FUNCTION_BLOCK MultiIOthersVlvStatus (* Composite Function Block Type *)
  (* Standard: 61499-2 *)
  (* Version 0.0, 8/28/2026, Schneider Electric, template *)
  PACKAGE SE.Nereda;
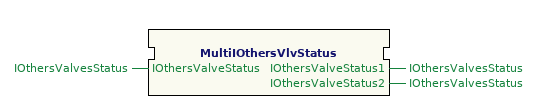
  SOCKETS
    IOthersValveStatus : IOthersValvesStatus;
  END_SOCKETS
  PLUGS
    IOthersValveStatus1 : IOthersValvesStatus;
    IOthersValveStatus2 : IOthersValvesStatus;
  END_PLUGS
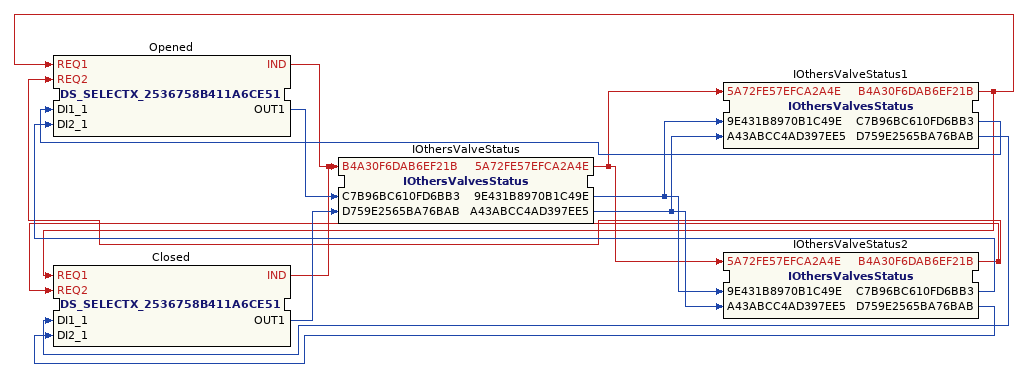
  FBS
    Opened : DS_SELECTX_2536758B411A6CE51; {SET_ATTRIBUTE(Configuration.GenericFBType.InterfaceParams, Runtime.Standard#CNTX:=2;CNTY:=1;DI${CNTX,_,CNTY$}:BOOL)}
    Closed : DS_SELECTX_2536758B411A6CE51; {SET_ATTRIBUTE(Configuration.GenericFBType.InterfaceParams, Runtime.Standard#CNTX:=2;CNTY:=1;DI${CNTX,_,CNTY$}:BOOL)}
  END_FBS
  EVENT_CONNECTIONS
    IOthersValveStatus.5A72FE57EFCA2A4E TO IOthersValveStatus1.5A72FE57EFCA2A4E;
    IOthersValveStatus.5A72FE57EFCA2A4E TO IOthersValveStatus2.5A72FE57EFCA2A4E;
    Opened.IND TO IOthersValveStatus.B4A30F6DAB6EF21B;
    Closed.IND TO IOthersValveStatus.B4A30F6DAB6EF21B;
    IOthersValveStatus1.B4A30F6DAB6EF21B TO Opened.REQ1;
    IOthersValveStatus2.B4A30F6DAB6EF21B TO Opened.REQ2;
    IOthersValveStatus1.B4A30F6DAB6EF21B TO Closed.REQ1;
    IOthersValveStatus2.B4A30F6DAB6EF21B TO Closed.REQ2;
  END_CONNECTIONS
  DATA_CONNECTIONS
    IOthersValveStatus.9E431B8970B1C49E TO IOthersValveStatus1.9E431B8970B1C49E;
    IOthersValveStatus.A43ABCC4AD397EE5 TO IOthersValveStatus1.A43ABCC4AD397EE5;
    IOthersValveStatus.9E431B8970B1C49E TO IOthersValveStatus2.9E431B8970B1C49E;
    IOthersValveStatus.A43ABCC4AD397EE5 TO IOthersValveStatus2.A43ABCC4AD397EE5;
    Opened.OUT1 TO IOthersValveStatus.C7B96BC610FD6BB3;
    Closed.OUT1 TO IOthersValveStatus.D759E2565BA76BAB;
    IOthersValveStatus1.C7B96BC610FD6BB3 TO Opened.DI1_1;
    IOthersValveStatus2.C7B96BC610FD6BB3 TO Opened.DI2_1;
    IOthersValveStatus1.D759E2565BA76BAB TO Closed.DI1_1;
    IOthersValveStatus2.D759E2565BA76BAB TO Closed.DI2_1;
  END_CONNECTIONS
END_FUNCTION_BLOCK
